(* IEC 61131-3 sources: beckhoffAutomationInterface/ST/Shark/Lib/ManualPanels, 6 files *)

(* ---- FB_DigitalInputManualPanel.st ---- *)
// Manual control panel for digital-input subsystem.
//
// Lib version — stateful FB; HMI binds to VAR fields directly.
FUNCTION_BLOCK FB_DigitalInputManualPanel
VAR_INPUT
    ipSubsystem : I_DigitalInputSubsystem;
    nMaxInput   : INT;
END_VAR
VAR
    // User Inputs (HMI)
    nSelectedInput  : INT := 1;

    // User Outputs (HMI)
    bSelectedState  : BOOL;
    bSelectedValid  : BOOL;
    bSubsystemValid : BOOL;
    bSubsystemReady : BOOL;

    ipSelectedInput : I_DigitalInput;
END_VAR

    IF ipSubsystem = 0 OR NOT ipSubsystem.IsInitialized() THEN
        bSubsystemReady := FALSE;
        bSubsystemValid := FALSE;
        bSelectedValid  := FALSE;
        bSelectedState  := FALSE;
        RETURN;
    END_IF

    bSubsystemReady := TRUE;
    bSubsystemValid := TRUE;
    ipSelectedInput := 0;
    bSelectedValid  := FALSE;

    IF nSelectedInput >= 1 AND nSelectedInput <= nMaxInput THEN
        ipSelectedInput := ipSubsystem.GetInputByIndex(nSelectedInput);
        bSelectedValid  := ipSelectedInput <> 0;
    END_IF

    IF ipSelectedInput <> 0 THEN
        bSelectedState := ipSelectedInput.GetState();
    ELSE
        bSelectedState := FALSE;
    END_IF

END_FUNCTION_BLOCK

(* ---- FB_DigitalOutputManualPanel.st ---- *)
// Manual control panel for digital-output subsystem.
//
// Lib version — stateful FB; HMI binds to VAR fields directly.
FUNCTION_BLOCK FB_DigitalOutputManualPanel
VAR_INPUT
    ipSubsystem : I_DigitalOutputSubsystem;
    nMaxOutput  : INT;
END_VAR
VAR
    // User Inputs (HMI)
    nSelectedOutput  : INT := 1;
    bCmdSetOn        : BOOL;
    bCmdSetOff       : BOOL;
    bCmdToggle       : BOOL;

    // User Outputs (HMI)
    bSelectedState   : BOOL;
    bSelectedValid   : BOOL;
    bLastCmdOk       : BOOL;
    bSubsystemReady  : BOOL;

    ipSelectedOutput : I_DigitalOutput;
END_VAR

    IF ipSubsystem = 0 OR NOT ipSubsystem.IsInitialized() THEN
        bSubsystemReady := FALSE;
        bSelectedValid  := FALSE;
        bSelectedState  := FALSE;
        bCmdSetOn       := FALSE;
        bCmdSetOff      := FALSE;
        bCmdToggle      := FALSE;
        RETURN;
    END_IF

    bSubsystemReady  := TRUE;
    ipSelectedOutput := 0;
    bSelectedValid   := FALSE;

    IF nSelectedOutput >= 1 AND nSelectedOutput <= nMaxOutput THEN
        ipSelectedOutput := ipSubsystem.GetOutputByIndex(nSelectedOutput);
        bSelectedValid   := ipSelectedOutput <> 0;
    END_IF

    IF NOT bSelectedValid OR ipSelectedOutput = 0 THEN
        bLastCmdOk     := FALSE;
        bSelectedState := FALSE;
        bCmdSetOn      := FALSE;
        bCmdSetOff     := FALSE;
        bCmdToggle     := FALSE;
        RETURN;
    END_IF

    bSelectedState := ipSelectedOutput.GetOutput();
    bLastCmdOk     := FALSE;

    IF bCmdSetOn THEN
        ipSelectedOutput.SetOutput(TRUE);
        bLastCmdOk := TRUE;
        bCmdSetOn  := FALSE;
    END_IF

    IF bCmdSetOff THEN
        ipSelectedOutput.SetOutput(FALSE);
        bLastCmdOk := TRUE;
        bCmdSetOff := FALSE;
    END_IF

    IF bCmdToggle THEN
        ipSelectedOutput.SetOutput(NOT bSelectedState);
        bLastCmdOk := TRUE;
        bCmdToggle := FALSE;
    END_IF

END_FUNCTION_BLOCK

(* ---- FB_FlowManualPanel.st ---- *)
// Manual control panel for flow subsystem.
//
// Lib version — stateful FB; HMI binds to VAR fields directly.
FUNCTION_BLOCK FB_FlowManualPanel
VAR_INPUT
    ipSubsystem : I_FlowSubsystem;
    nMaxZone    : INT;
END_VAR
VAR
    // User Inputs (HMI)
    nSelectedZone        : INT := 1;
    rSelectedSetpoint    : LREAL := 0.0;
    bCmdApplySetpoint    : BOOL;
    bCmdEnable           : BOOL;
    bCmdDisable          : BOOL;
    bCmdReset            : BOOL;

    // User Outputs (HMI)
    stSelectedStatus     : ST_ControllerStatus;
    bLastCmdOk           : BOOL;
    bSelectedZoneValid   : BOOL;
    bSubsystemAnyError   : BOOL;
    bSubsystemReady      : BOOL;

    ipSelectedController : I_Controller;
END_VAR

    IF ipSubsystem = 0 OR NOT ipSubsystem.IsInitialized() THEN
        bSubsystemReady    := FALSE;
        bSubsystemAnyError := FALSE;
        bSelectedZoneValid := FALSE;
        bCmdApplySetpoint  := FALSE;
        bCmdEnable         := FALSE;
        bCmdDisable        := FALSE;
        bCmdReset          := FALSE;
        RETURN;
    END_IF

    bSubsystemReady    := TRUE;
    bSubsystemAnyError := ipSubsystem.HasAnyError();

    ipSelectedController := 0;
    bSelectedZoneValid   := FALSE;

    IF nSelectedZone >= 1 AND nSelectedZone <= nMaxZone THEN
        ipSelectedController := ipSubsystem.GetControllerByIndex(nSelectedZone);
        bSelectedZoneValid   := ipSelectedController <> 0;
    END_IF

    IF ipSelectedController = 0 THEN
        bLastCmdOk                        := FALSE;
        bCmdApplySetpoint                 := FALSE;
        bCmdEnable                        := FALSE;
        bCmdDisable                       := FALSE;
        bCmdReset                         := FALSE;
        stSelectedStatus.rMeasuredValue   := 0.0;
        stSelectedStatus.rSetpoint        := 0.0;
        stSelectedStatus.rOutput          := 0.0;
        stSelectedStatus.bEnabled         := FALSE;
        stSelectedStatus.bAtSetpoint      := FALSE;
        stSelectedStatus.stError.eErrorId := E_ErrorId.NO_ERROR;
        stSelectedStatus.stError.sSource  := '';
        stSelectedStatus.stError.sMessage := '';
        RETURN;
    END_IF

    stSelectedStatus := ipSelectedController.GetStatus();
    bLastCmdOk       := FALSE;

    IF bCmdApplySetpoint THEN
        bLastCmdOk        := ipSelectedController.SetSetpoint(rSelectedSetpoint);
        bCmdApplySetpoint := FALSE;
    END_IF

    IF bCmdDisable THEN
        bLastCmdOk  := ipSelectedController.Enable(FALSE);
        bCmdDisable := FALSE;
        bCmdEnable  := FALSE;
    ELSIF bCmdEnable THEN
        bLastCmdOk := ipSelectedController.Enable(TRUE);
        bCmdEnable := FALSE;
    END_IF

    IF bCmdReset THEN
        bLastCmdOk := ipSelectedController.Reset();
        bCmdReset  := FALSE;
    END_IF

END_FUNCTION_BLOCK

(* ---- FB_PressureManualPanel.st ---- *)
// Manual control panel for pressure subsystem.
//
// Lib version — stateful FB; HMI binds to VAR fields directly.
// Switches between sensor view and controller view via bViewSensor.
FUNCTION_BLOCK FB_PressureManualPanel
VAR_INPUT
    ipSubsystem : I_PressureSubsystem;
    nMaxSensor  : INT;
    nMaxCtrl    : INT;
END_VAR
VAR
    // Mode Selection
    bViewSensor          : BOOL := TRUE;   // TRUE = sensor view, FALSE = controller view

    // User Inputs (HMI)
    nSelectedSensor      : INT := 1;
    nSelectedController  : INT := 1;
    rSelectedSetpoint    : LREAL := 0.0;
    bCmdApplySetpoint    : BOOL;
    bCmdEnable           : BOOL;
    bCmdDisable          : BOOL;
    bCmdReset            : BOOL;

    // Outputs
    stSelectedStatus     : ST_ControllerStatus;
    bLastCmdOk           : BOOL;
    bSelectedValid       : BOOL;
    bSubsystemAnyError   : BOOL;
    bSubsystemReady      : BOOL;

    ipSelectedSensor     : I_Sensor;
    ipSelectedController : I_Controller;
END_VAR

    IF ipSubsystem = 0 OR NOT ipSubsystem.IsInitialized() THEN
        bSubsystemReady    := FALSE;
        bSubsystemAnyError := FALSE;
        bSelectedValid     := FALSE;
        bCmdApplySetpoint  := FALSE;
        bCmdEnable         := FALSE;
        bCmdDisable        := FALSE;
        bCmdReset          := FALSE;
        RETURN;
    END_IF

    bSubsystemReady    := TRUE;
    bSubsystemAnyError := ipSubsystem.HasAnyError();

    ipSelectedSensor     := 0;
    ipSelectedController := 0;
    bSelectedValid       := FALSE;

    IF bViewSensor THEN
        IF nSelectedSensor >= 1 AND nSelectedSensor <= nMaxSensor THEN
            ipSelectedSensor := ipSubsystem.GetSensorByIndex(nSelectedSensor);
            bSelectedValid   := ipSelectedSensor <> 0;
        END_IF
    ELSE
        IF nSelectedController >= 1 AND nSelectedController <= nMaxCtrl THEN
            ipSelectedController := ipSubsystem.GetControllerByIndex(nSelectedController);
            bSelectedValid       := ipSelectedController <> 0;
        END_IF
    END_IF

    IF ipSelectedSensor <> 0 THEN
        stSelectedStatus.rMeasuredValue := ipSelectedSensor.GetMeasurement();
        stSelectedStatus.rSetpoint      := 0.0;
        stSelectedStatus.rOutput        := 0.0;
        stSelectedStatus.bEnabled       := TRUE;
        stSelectedStatus.bAtSetpoint    := FALSE;
        stSelectedStatus.stError        := ipSelectedSensor.GetError();
    ELSIF ipSelectedController <> 0 THEN
        stSelectedStatus := ipSelectedController.GetStatus();
    ELSE
        stSelectedStatus.rMeasuredValue   := 0.0;
        stSelectedStatus.rSetpoint        := 0.0;
        stSelectedStatus.rOutput          := 0.0;
        stSelectedStatus.bEnabled         := FALSE;
        stSelectedStatus.bAtSetpoint      := FALSE;
        stSelectedStatus.stError.eErrorId := E_ErrorId.NO_ERROR;
        stSelectedStatus.stError.sSource  := '';
        stSelectedStatus.stError.sMessage := '';
    END_IF

    IF bViewSensor OR ipSelectedController = 0 THEN
        bLastCmdOk        := FALSE;
        bCmdApplySetpoint := FALSE;
        bCmdEnable        := FALSE;
        bCmdDisable       := FALSE;
        bCmdReset         := FALSE;
        RETURN;
    END_IF

    bLastCmdOk := FALSE;

    IF bCmdApplySetpoint THEN
        bLastCmdOk        := ipSelectedController.SetSetpoint(rSelectedSetpoint);
        bCmdApplySetpoint := FALSE;
    END_IF

    IF bCmdDisable THEN
        bLastCmdOk  := ipSelectedController.Enable(FALSE);
        bCmdDisable := FALSE;
        bCmdEnable  := FALSE;
    ELSIF bCmdEnable THEN
        bLastCmdOk := ipSelectedController.Enable(TRUE);
        bCmdEnable := FALSE;
    END_IF

    IF bCmdReset THEN
        bLastCmdOk := ipSelectedController.Reset();
        bCmdReset  := FALSE;
    END_IF

END_FUNCTION_BLOCK

(* ---- FB_TemperatureManualPanel.st ---- *)
// Manual control panel for temperature subsystem.
//
// Lib version — stateful FB; HMI binds to VAR fields directly.
// Default setpoint is 0.0; caller can override via rSelectedSetpoint VAR field.
FUNCTION_BLOCK FB_TemperatureManualPanel
VAR_INPUT
    ipSubsystem : I_TemperatureSubsystem;
    nMaxZone    : INT;
END_VAR
VAR
    // User Inputs - Selection
    nSelectedZone           : INT := 1;
    bSelectWholeZone        : BOOL := TRUE;   // TRUE = control whole zone, FALSE = single channel
    nSelectedChannelIdx     : INT := 1;       // 1..nSelectedZoneChannelCount (channel mode)
    rSelectedSetpoint       : LREAL := 0.0;
    bCmdApplySetpoint       : BOOL;
    bCmdEnable              : BOOL;
    bCmdDisable             : BOOL;
    bCmdReset               : BOOL;

    // User Outputs
    stSelectedStatus        : ST_ControllerStatus;
    bLastCmdOk              : BOOL;
    bSelectedValid          : BOOL;
    bIsControllable         : BOOL;
    nSelectedZoneChannelCount : INT;          // channels in the selected zone (HMI bound)
    bSubsystemAnyError      : BOOL;
    bSubsystemAllAtSetpoint : BOOL;
    bSubsystemReady         : BOOL;
    stFirstError            : ST_Error;

    ipSelectedSensor     : I_Sensor;
    ipSelectedController : I_Controller;
END_VAR

    IF ipSubsystem = 0 OR NOT ipSubsystem.IsInitialized() THEN
        bSubsystemReady         := FALSE;
        bSubsystemAnyError      := FALSE;
        bSubsystemAllAtSetpoint := FALSE;
        bSelectedValid          := FALSE;
        bIsControllable         := FALSE;
        nSelectedZoneChannelCount := 0;
        stFirstError.eErrorId   := E_ErrorId.NO_ERROR;
        bCmdApplySetpoint       := FALSE;
        bCmdEnable              := FALSE;
        bCmdDisable             := FALSE;
        bCmdReset               := FALSE;
        RETURN;
    END_IF

    bSubsystemReady         := TRUE;
    bSubsystemAnyError      := ipSubsystem.HasAnyError();
    bSubsystemAllAtSetpoint := ipSubsystem.AllAtSetpoint();
    stFirstError            := ipSubsystem.GetFirstError();

    ipSelectedSensor     := 0;
    ipSelectedController := 0;
    bSelectedValid       := FALSE;
    bIsControllable      := FALSE;
    nSelectedZoneChannelCount := 0;

    IF nSelectedZone >= 1 AND nSelectedZone <= nMaxZone THEN
        nSelectedZoneChannelCount := ipSubsystem.GetChannelCountByIndex(nSelectedZone);
        IF bSelectWholeZone THEN
            ipSelectedSensor     := ipSubsystem.GetTemperatureByIndex(nSelectedZone);
            ipSelectedController := ipSubsystem.GetControllerByIndex(nSelectedZone);
        ELSE
            ipSelectedController := ipSubsystem.GetChannelControllerByZoneIndex(nSelectedZone, nSelectedChannelIdx);
        END_IF
    END_IF

    bSelectedValid  := (ipSelectedSensor <> 0) OR (ipSelectedController <> 0);
    bIsControllable := ipSelectedController <> 0;

    IF ipSelectedController <> 0 THEN
        stSelectedStatus := ipSelectedController.GetStatus();
    ELSIF ipSelectedSensor <> 0 THEN
        stSelectedStatus.rMeasuredValue := ipSelectedSensor.GetMeasurement();
        stSelectedStatus.rSetpoint      := 0.0;
        stSelectedStatus.rOutput        := 0.0;
        stSelectedStatus.bEnabled       := FALSE;
        stSelectedStatus.bAtSetpoint    := FALSE;
        stSelectedStatus.stError        := ipSelectedSensor.GetError();
    ELSE
        stSelectedStatus.rMeasuredValue   := 0.0;
        stSelectedStatus.rSetpoint        := 0.0;
        stSelectedStatus.rOutput          := 0.0;
        stSelectedStatus.bEnabled         := FALSE;
        stSelectedStatus.bAtSetpoint      := FALSE;
        stSelectedStatus.stError.eErrorId := E_ErrorId.NO_ERROR;
        stSelectedStatus.stError.sSource  := '';
        stSelectedStatus.stError.sMessage := '';
    END_IF

    IF ipSelectedController = 0 THEN
        bCmdApplySetpoint := FALSE;
        bCmdEnable        := FALSE;
        bCmdDisable       := FALSE;
        bCmdReset         := FALSE;
        RETURN;
    END_IF

    bLastCmdOk := FALSE;

    IF bCmdApplySetpoint THEN
        bLastCmdOk        := ipSelectedController.SetSetpoint(rSelectedSetpoint);
        bCmdApplySetpoint := FALSE;
    END_IF

    IF bCmdDisable THEN
        bLastCmdOk  := ipSelectedController.Enable(FALSE);
        bCmdDisable := FALSE;
        bCmdEnable  := FALSE;
    ELSIF bCmdEnable THEN
        bLastCmdOk := ipSelectedController.Enable(TRUE);
        bCmdEnable := FALSE;
    END_IF

    IF bCmdReset THEN
        bLastCmdOk := ipSelectedController.Reset();
        bCmdReset  := FALSE;
    END_IF

END_FUNCTION_BLOCK

(* ---- FB_ValveManualPanel.st ---- *)
// Manual control panel for valve subsystem.
//
// Lib version — stateful FB; HMI binds to VAR fields directly.
// Subsystem is injected via the interface; max-id is supplied by the caller.
FUNCTION_BLOCK FB_ValveManualPanel
VAR_INPUT
    ipSubsystem : I_ValveSubsystem;
    nMaxValveId : INT;
END_VAR
VAR
    // User Inputs (HMI)
    nSelectedValveId    : INT := 1;
    bCmdOpen            : BOOL;
    bCmdClose           : BOOL;
    bCmdReset           : BOOL;

    // User Outputs (HMI)
    bLastCmdOk          : BOOL;
    bSelectedValveValid : BOOL;
    bIsOpen             : BOOL;
    bSubsystemAnyError  : BOOL;
    bSubsystemReady     : BOOL;

    ipSelectedValve     : I_Valve;
END_VAR

    IF ipSubsystem = 0 OR NOT ipSubsystem.IsInitialized() THEN
        bSubsystemReady     := FALSE;
        bSubsystemAnyError  := FALSE;
        bSelectedValveValid := FALSE;
        bIsOpen             := FALSE;
        bLastCmdOk          := FALSE;
        bCmdOpen            := FALSE;
        bCmdClose           := FALSE;
        bCmdReset           := FALSE;
        RETURN;
    END_IF

    bSubsystemReady    := TRUE;
    bSubsystemAnyError := ipSubsystem.HasAnyError();

    ipSelectedValve     := 0;
    bSelectedValveValid := FALSE;

    IF nSelectedValveId >= 1 AND nSelectedValveId <= nMaxValveId THEN
        ipSelectedValve     := ipSubsystem.GetValveByIndex(nSelectedValveId);
        bSelectedValveValid := ipSelectedValve <> 0;
    END_IF

    IF ipSelectedValve = 0 THEN
        bIsOpen    := FALSE;
        bLastCmdOk := FALSE;
        bCmdOpen   := FALSE;
        bCmdClose  := FALSE;
        bCmdReset  := FALSE;
        RETURN;
    END_IF

    bIsOpen    := ipSelectedValve.IsOpen();
    bLastCmdOk := FALSE;

    IF bCmdOpen THEN
        ipSelectedValve.Open();
        bLastCmdOk := TRUE;
        bCmdOpen   := FALSE;
    END_IF

    IF bCmdClose THEN
        ipSelectedValve.Close();
        bLastCmdOk := TRUE;
        bCmdClose  := FALSE;
    END_IF

    IF bCmdReset THEN
        ipSelectedValve.Reset();
        bLastCmdOk := TRUE;
        bCmdReset  := FALSE;
    END_IF

END_FUNCTION_BLOCK
